FUNCTION_BLOCK ASE_TRANSFER_CN (* Composite Function Block Type *)
  (* Standard: 61499-2 *)
  (* Version 0.2, 2003-12-05, JHC, Rockwell Automation, Renamed from NEWCOMPFB. *)
  (* Version 0.1, 2002-01-08, JHC, Rockwell Automation, Added DLY FB as example. *)
  (* Version 0.0, 2000-05-27, JHC, Rockwell Automation *)
  (* Compiler header: package fb.rt.student; *)
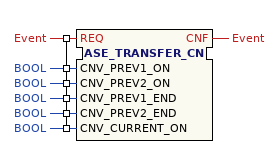
  EVENT_INPUT
    REQ WITH CNV_PREV1_ON, CNV_PREV2_ON, CNV_PREV1_END, CNV_PREV2_END, CNV_CURRENT_ON; (* Normal Execution Request *)
  END_EVENT
  EVENT_OUTPUT
    CNF; (* Execution Confirmation *)
  END_EVENT
  VAR_INPUT
    CNV_PREV1_ON : BOOL;
    CNV_PREV2_ON : BOOL;
    CNV_PREV1_END : BOOL;
    CNV_PREV2_END : BOOL;
    CNV_CURRENT_ON : BOOL;
  END_VAR
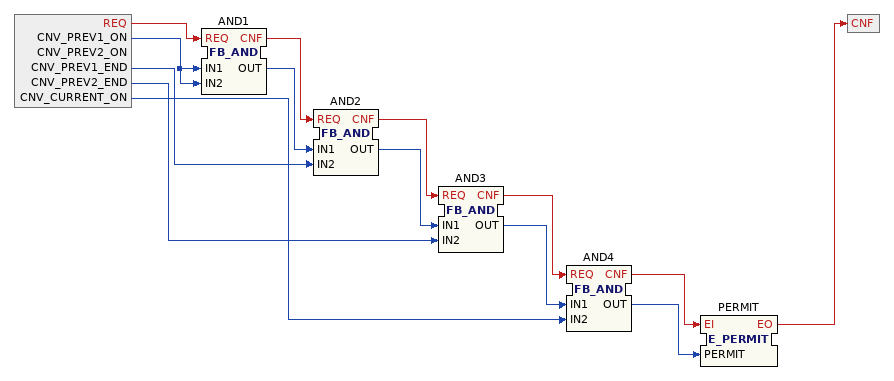
  FBS
    AND1 : FB_AND;
    AND2 : FB_AND;
    AND3 : FB_AND;
    AND4 : FB_AND;
    PERMIT : E_PERMIT;
  END_FBS
  EVENT_CONNECTIONS
    REQ TO AND1.REQ;
    AND1.CNF TO AND2.REQ;
    AND2.CNF TO AND3.REQ;
    REQ TO AND1.REQ;
    AND1.CNF TO AND2.REQ;
    AND2.CNF TO AND3.REQ;
    AND3.CNF TO AND4.REQ;
    AND4.CNF TO PERMIT.EI;
    PERMIT.EO TO CNF;
  END_CONNECTIONS
  DATA_CONNECTIONS
    AND1.OUT TO AND2.IN1;
    AND2.OUT TO AND3.IN1;
    CNV_PREV1_ON TO AND1.IN1;
    CNV_PREV1_ON TO AND1.IN2;
    CNV_PREV1_END TO AND2.IN2;
    CNV_PREV2_END TO AND3.IN2;
    AND1.OUT TO AND2.IN1;
    AND2.OUT TO AND3.IN1;
    CNV_PREV1_ON TO AND1.IN1;
    CNV_PREV1_ON TO AND1.IN2;
    CNV_PREV1_END TO AND2.IN2;
    CNV_PREV2_END TO AND3.IN2;
    AND3.OUT TO AND4.IN1;
    AND4.OUT TO PERMIT.PERMIT;
    CNV_CURRENT_ON TO AND4.IN2;
  END_CONNECTIONS
END_FUNCTION_BLOCK
